PROGRAM MAIN
VAR
END_VAR

END_PROGRAM

(* stored: Version 1.1.0.1
   POU MAIN: Id {f13ba1f9-b9cc-488a-aba1-9ee71a387b30} *)
